(* CODESYS project AgitatorMotor.xml

Project tree, tasks and I/O mapping:
  function block AgitatorMotor [LD]
*)

// AgitatorMotor
FUNCTION_BLOCK AgitatorMotor
VAR_INPUT
	Forward: BOOL;
	Reverse: BOOL;
	Settings: MotorSettings;
END_VAR
VAR_OUTPUT
	MotorOutput: BOOL;
	ReverseOutput: BOOL;
	SpeedOutput: UINT;
END_VAR
VAR
END_VAR

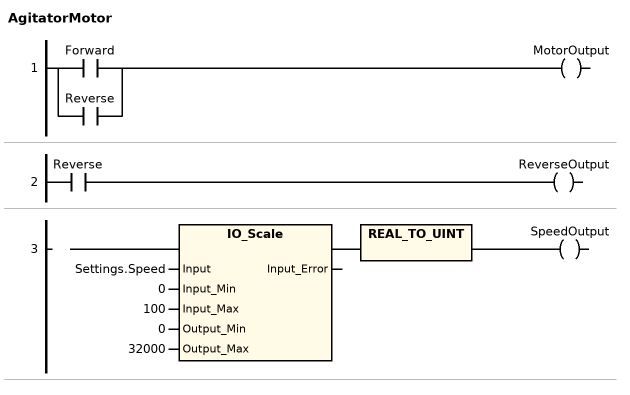
// NETWORK 1
MotorOutput := Forward OR Reverse;

// NETWORK 2
ReverseOutput := Reverse;

// NETWORK 3
SpeedOutput := REAL_TO_UINT(IO_Scale(Input := Settings.Speed, Input_Min := 0, Input_Max := 100, Output_Min := 0, Output_Max := 32000));

END_FUNCTION_BLOCK
